Yaskawa INFORM job: CLOSE-CURTAIN.JBI

/JOB
//NAME CLOSE-CURTAIN
//POS
///NPOS 0,0,0,0,0,0
//INST
///DATE 2018/08/30 13:35
///ATTR SC,RW
NOP
DOUT OT#(5) OFF
TIMER T=0.20
DOUT OT#(15) ON
WAIT IN#(16)=ON T=15.00
*error
IFTHEN IN#(16)=OFF
	 SETUALM 8000 "Curtain is not closed" 0
	 PAUSE
	 JUMP *error
ENDIF
*1
DOUT OT#(15) OFF
DOUT OT#(5) OFF
*END
END
